FUNCTION_BLOCK C_SQLCLIENT EXTENDS C_DBADAPTOR
VAR_INPUT
END_VAR
VAR_OUTPUT
END_VAR
VAR
	_FBADDCONN		: FB_DBConnectionAdd;
	//_FBSQLDELETE 	: FB_DBRecordDelete;
	_FBSQLINSERT 	: FB_DBRecordInsert_EX;
	_FBSQLSELECT 	: FB_DBRecordArraySelect;
END_VAR

{attribute 'object_name' := 'SQL_EXECUTE_NONQUERY'}
METHOD SQL_EXECUTE_NONQUERY : DINT
VAR_INPUT
	SQL : POINTER TO T_SQL_COMMAND;
END_VAR
_FBSQLINSERT(
	sNetID:= sAmsNetId, 
	hDBID:= DB_ID, 
	pCmdAddr:= SQL, 
	cbCmdSize:= GET_SQL_COMMAND_LENGTH(SQL), 
	bExecute:= TRUE, 
	tTimeout:= _TIMEOUT );
IF _FBSQLINSERT.bError THEN
	_FBSQLINSERT(bExecute:= FALSE);
	SQL_EXECUTE_NONQUERY := 1;
	RETURN;
ELSIF NOT _FBSQLINSERT.bBusy THEN
	_FBSQLINSERT(bExecute:= FALSE);
	SQL_EXECUTE_NONQUERY := -1;
	RETURN;
ELSE
	SQL_EXECUTE_NONQUERY := 0;
	RETURN;
END_IF
END_METHOD

{attribute 'object_name' := 'SQL_EXECUTE_QUERY'}
METHOD SQL_EXECUTE_QUERY : DINT
VAR_INPUT
	SQL_PTR				: POINTER TO T_SQL_COMMAND;
	START_INDEX			: UDINT;
	ROWS_TO_READ		: UDINT;
	PTR_DATA_OUT		: PVOID;
	DATA_SIZE			: UDINT;
	DATABASE_ROWS		: POINTER TO UDINT;
END_VAR
_FBSQLSELECT(
	sNetID:= sAmsNetId, 
	hDBID:= DB_ID, 
	pCmdAddr:= SQL_PTR, 
	cbCmdSize:= GET_SQL_COMMAND_LENGTH(SQL_PTR), 
	nStartIndex:= START_INDEX, 
	nRecordCount:= ROWS_TO_READ, 
	pDestAddr:= PTR_DATA_OUT, 
	cbRecordArraySize:= DATA_SIZE, 
	bExecute:= TRUE, 
	tTimeout:= _TIMEOUT );
IF _FBSQLSELECT.bError THEN
	_FBSQLSELECT(bExecute:= FALSE);
	SQL_EXECUTE_QUERY := 1;
	RETURN;
ELSIF NOT _FBSQLSELECT.bBusy THEN
	DATABASE_ROWS^ := _FBSQLSELECT.nRecords;
	_FBSQLSELECT(bExecute:= FALSE);
	SQL_EXECUTE_QUERY := -1;
	RETURN;
ELSE 
	SQL_EXECUTE_QUERY := 0;
	RETURN;
END_IF
END_METHOD

METHOD CREATE_CONNECTION : DINT
VAR_INPUT
	URL					: STRING(255);
	TABLE				: STRING(255);
	NAME				: STRING(255);
	Database_Handle_Out : POINTER TO UDINT;	
END_VAR
_FBADDCONN(
	sNetID:= sAmsNetId, 
	eDBType:= eDBType_SQLite, 
	eDBValueType:= eDBValue_Bytes, 
	sDBServer:= NAME, 
	sDBUrl:= URL, 
	sDBTable:= TABLE, 
	bExecute:= TRUE, 
	tTimeout:= _TIMEOUT, 
	bBusy=> , 
	bError=> , 
	nErrID=> , 
	hDBID=> );
IF _FBADDCONN.bError THEN
	_FBADDCONN(bExecute:= FALSE);
	CREATE_CONNECTION := 1;
	RETURN; 
ELSIF NOT _FBADDCONN.bBusy THEN
	Database_Handle_Out^ := _FBADDCONN.hDBID;
	_FBADDCONN(bExecute:= FALSE);
	CREATE_CONNECTION := -1;
	RETURN; 
ELSE
	CREATE_CONNECTION := 0;
	RETURN;
END_IF
END_METHOD

END_FUNCTION_BLOCK

(* stored: Version 1.1.0.1, ProductVersion 3.1.4020.3
   POU C_SQLITE: Id {a7ee5403-6d43-4885-8669-cfa9297b2c15}, SpecialFunc None
   Folder METHODS: Id {e654c67b-c57e-4f3d-a34c-33451736c15b}
   Folder SQL: Id {a1eb873f-d914-4db2-ae6d-e7813fe3a398}
   Method SQL_EXECUTE_NONQUERY: Id {813d7971-78c7-4d45-8f56-becb63644dad}
   Method SQL_EXECUTE_QUERY: Id {878a5881-e6d5-4326-bd4d-c9c7cade3cd3}
   Method CREATE_CONNECTION: Id {a87967c6-5945-4b2d-b200-fc867ecb11b3} *)
